(* PLC project Unnamed, Unknown Unnamed 1 *)
(* stored: creationDateTime 2023-09-22T09:24:15, modificationDateTime 2023-09-28T21:40:20 *)

PROGRAM program3
  VAR
    FactoryIOReset0 AT %IX100.0 : BOOL;
    StartButton0 AT %IX100.1 : BOOL;
    EStop0 AT %IX100.2 : BOOL;
    Retro0 AT %IX100.3 : BOOL;
    Retro1 AT %IX100.4 : BOOL;
    VS00 AT %IX100.5 : BOOL;
    VS01 AT %IX100.6 : BOOL;
    VS02 AT %IX100.7 : BOOL;
    VS03 AT %IX101.0 : BOOL;
    TAPP0_Detected AT %IX101.1 : BOOL;
    TAPP0_MovingX AT %IX101.2 : BOOL;
    TAPP0_MovingZ AT %IX101.3 : BOOL;
    TAPP0_Rotating AT %IX101.4 : BOOL;
    Retro2 AT %IX101.5 : BOOL;
    RetroreflectiveSensor3 AT %IX101.6 : BOOL;
    Retro4 AT %IX101.7 : BOOL;
    VS10 AT %IX102.0 : BOOL;
    VS11 AT %IX102.1 : BOOL;
    VS12 AT %IX102.2 : BOOL;
    VisionSensor13 AT %IX102.3 : BOOL;
    TAPP1_Detected AT %IX102.4 : BOOL;
    TwoAxisPickPlace1_MovingX AT %IX102.5 : BOOL;
    TwoAxisPickPlace1_MovingZ AT %IX102.6 : BOOL;
    TwoAxisPickPlace1_Rotating AT %IX102.7 : BOOL;
    RetroreflectiveSensor5 AT %IX103.0 : BOOL;
    RetroreflectiveSensor6 AT %IX103.1 : BOOL;
    Retro7 AT %IX103.2 : BOOL;
    VS20 AT %IX103.3 : BOOL;
    VS21 AT %IX103.4 : BOOL;
    VS22 AT %IX103.5 : BOOL;
    VisionSensor23 AT %IX103.6 : BOOL;
    TAPP2_Detected AT %IX103.7 : BOOL;
    TwoAxisPickPlace2_MovingX AT %IX104.0 : BOOL;
    TwoAxisPickPlace2_MovingZ AT %IX104.1 : BOOL;
    TwoAxisPickPlace2_Rotating AT %IX104.2 : BOOL;
    RetroreflectiveSensor8 AT %IX104.3 : BOOL;
    RetroreflectiveSensor9 AT %IX104.4 : BOOL;
    RetroreflectiveSensor10 AT %IX104.5 : BOOL;
    VisionSensor30 AT %IX104.6 : BOOL;
    VisionSensor31 AT %IX104.7 : BOOL;
    VisionSensor32 AT %IX105.0 : BOOL;
    VisionSensor33 AT %IX105.1 : BOOL;
    Retro11 AT %IX105.2 : BOOL;
    Retro12 AT %IX105.3 : BOOL;
    Retro13 AT %IX105.4 : BOOL;
    Retro14 AT %IX105.5 : BOOL;
    Retro15 AT %IX105.6 : BOOL;
    Retro16 AT %IX105.7 : BOOL;
    TAPP0X AT %QX100.0 : BOOL;
    TAPP0Z AT %QX100.1 : BOOL;
    TAPP0_Grab AT %QX100.2 : BOOL;
    TAPP0_RotateCW AT %QX100.3 : BOOL;
    TAPP0_RotateCCW AT %QX100.4 : BOOL;
    BC_6m_0 AT %QX100.5 : BOOL;
    BC_6m_1 AT %QX100.6 : BOOL;
    BC_6m_2 AT %QX100.7 : BOOL;
    BC_6m_3 AT %QX101.0 : BOOL;
    BC_6m_4 AT %QX101.1 : BOOL;
    TAPP1X AT %QX101.2 : BOOL;
    TAPP1Z AT %QX101.3 : BOOL;
    TAPP1_Grab AT %QX101.4 : BOOL;
    TAPP1_RotateCCW AT %QX101.5 : BOOL;
    TAPP1_RotateCW AT %QX101.6 : BOOL;
    GreenBoxDetected AT %QX101.7 : BOOL;
    TAPP2X AT %QX102.0 : BOOL;
    TAPP2Z AT %QX102.1 : BOOL;
    TAPP2_Grab AT %QX102.2 : BOOL;
    TAPP2_RotateCW AT %QX102.3 : BOOL;
    TAPP2_RotateCCW AT %QX102.4 : BOOL;
    BC_2m_0 AT %QX102.5 : BOOL;
    BlueBoxDetected AT %QX102.6 : BOOL;
    GreyBoxDetected0 AT %QX102.7 : BOOL;
    StackLight0_Green AT %QX103.0 : BOOL;
    StackLight0_Yellow AT %QX103.1 : BOOL;
    StackLight0_Red AT %QX103.2 : BOOL;
    StackLight1_Green AT %QX103.3 : BOOL;
    StackLight1_Yellow AT %QX103.4 : BOOL;
    StackLight1_Red AT %QX103.5 : BOOL;
    StackLight2_Green AT %QX103.6 : BOOL;
    StackLight2_Yellow AT %QX103.7 : BOOL;
    StackLight2_Red AT %QX104.0 : BOOL;
    LightIndicator_Red_2 AT %QX104.1 : BOOL;
    BlueGrabbed AT %QW100 : INT;
    GreenGrabbed AT %QW101 : INT;
    GreyGrabbed AT %QW102 : INT;
    BlueMissed AT %QW103 : INT;
    GreenMissed AT %QW104 : INT;
    GreyMissed AT %QW105 : INT;
  END_VAR
  VAR
    FactoryReset : BOOL;
    StartCondition : BOOL;
    RS1 : RS;
    TAPP0ZPT : TIME := T#2s;
    RCW0PT : TIME := T#2s;
    RCW1PT : TIME := T#2s;
    RCW2PT : TIME := T#2s;
    TAPP1ZPT : TIME := T#2s;
    TAPP2ZPT : TIME := T#2s;
    TAPP0ZET : TIME;
    TAPP1ZET : TIME;
    TAPP2ZET : TIME;
    Grab0PT : TIME := T#0.5s;
    Grab2PT : TIME := T#0.5s;
    Grab1PT : TIME := T#0.5s;
    Grab0ET : TIME;
    RCW0ET : TIME;
    RCW1ET : TIME;
    RCW2ET : TIME;
    Grab1ET : TIME;
    Grab2ET : TIME;
    Grab0TPPT : TIME := T#3s;
    Grab1TPPT : TIME := T#3s;
    Grab2TPPT : TIME := T#3s;
    Grab0TPET : TIME;
    Grab1TPET : TIME;
    Grab2TPET : TIME;
    GreyBox : BOOL;
    RS5 : RS;
    GrabbedMax : INT := 50;
    RS11 : RS;
    RS9 : RS;
    RS10 : RS;
    RS12 : RS;
    TON0 : TON;
    RS14 : RS;
    TON1 : TON;
    RS15 : RS;
    RS16 : RS;
    TON2 : TON;
    TP0 : TP;
    RS13 : RS;
    RS17 : RS;
    RS18 : RS;
    RS2 : RS;
    CTU0 : CTU;
    RS20 : RS;
    CTU1 : CTU;
    RS21 : RS;
    CTU2 : CTU;
    RS30 : RS;
    CTU3 : CTU;
    RS31 : RS;
    RS32 : RS;
    RS7 : RS;
    RS37 : RS;
    RS38 : RS;
    TON8 : TON;
    CTU4 : CTU;
    RS41 : RS;
    CTU5 : CTU;
    RS42 : RS;
    RS19 : RS;
    RS22 : RS;
    RS23 : RS;
    RS24 : RS;
    RS25 : RS;
    TON3 : TON;
    RS6 : RS;
    RS26 : RS;
    RS27 : RS;
    TON4 : TON;
    TP1 : TP;
    TON5 : TON;
    RS28 : RS;
    RS29 : RS;
    RS33 : RS;
    RS34 : RS;
    RS35 : RS;
    RS36 : RS;
    TON6 : TON;
    TP2 : TP;
    TON7 : TON;
    RS43 : RS;
    RS44 : RS;
  END_VAR
  VAR  (* added by the conversion: wires and edge detectors of the diagram *)
    R_TRIG1 : R_TRIG;
    F_TRIG2 : F_TRIG;
    F_TRIG3 : F_TRIG;
    R_TRIG4 : R_TRIG;
    R_TRIG5 : R_TRIG;
    F_TRIG6 : F_TRIG;
    R_TRIG7 : R_TRIG;
    R_TRIG8 : R_TRIG;
    F_TRIG9 : F_TRIG;
    R_TRIG10 : R_TRIG;
    R_TRIG11 : R_TRIG;
  END_VAR

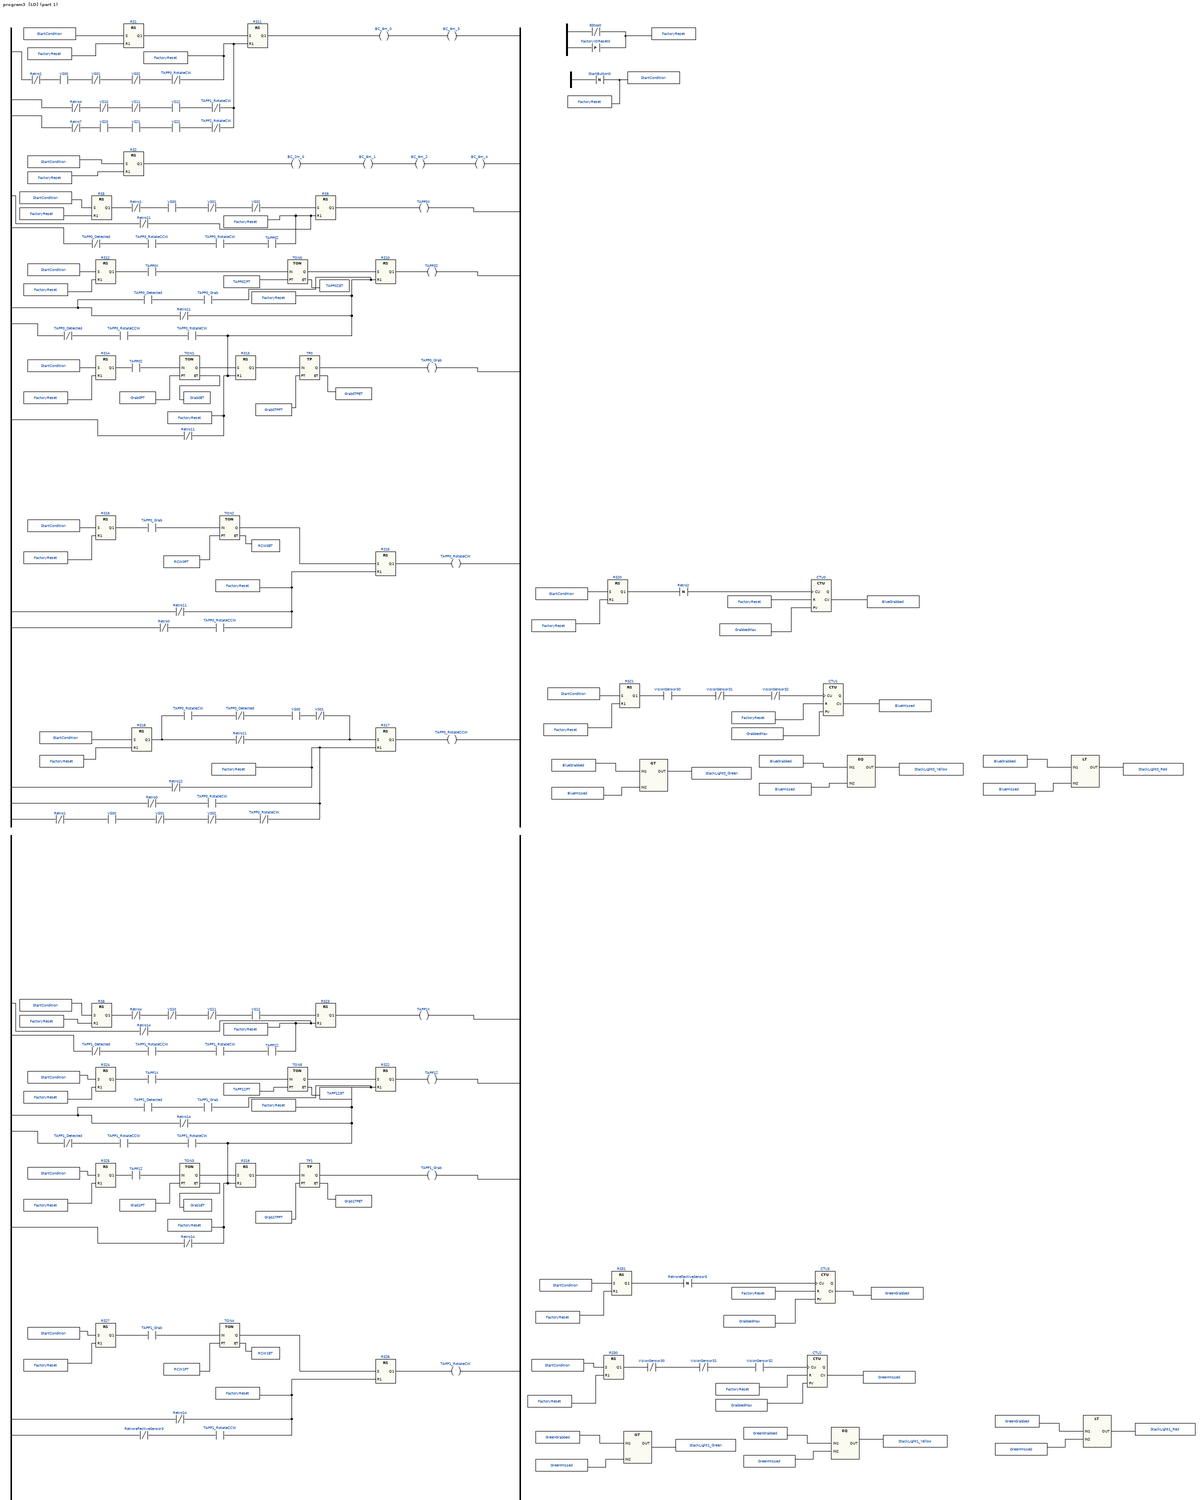
(* LD diagram, written out as Structured Text *)
R_TRIG1(CLK := FactoryIOReset0);
FactoryReset := NOT EStop0 OR R_TRIG1.Q;
RS1(S := StartCondition, R1 := FactoryReset);
RS11(S := RS1.Q1, R1 := FactoryReset OR NOT Retro1 AND VS00 AND NOT VS01 AND NOT VS02 AND NOT TAPP0_RotateCW OR NOT Retro4 AND NOT VS10 AND NOT VS11 AND VS12 AND NOT TAPP1_RotateCW OR NOT Retro7 AND VS20 AND VS21 AND VS22 AND NOT TAPP2_RotateCW);
BC_6m_0 := RS11.Q1;
BC_6m_3 := RS11.Q1;
F_TRIG2(CLK := StartButton0);
StartCondition := F_TRIG2.Q OR FactoryReset;
RS2(S := StartCondition, R1 := FactoryReset);
BC_2m_0 := RS2.Q1;
BC_6m_1 := RS2.Q1;
BC_6m_2 := RS2.Q1;
BC_6m_4 := RS2.Q1;
RS5(S := StartCondition, R1 := FactoryReset);
RS9(S := RS5.Q1 AND NOT Retro1 AND VS00 AND NOT VS01 AND NOT VS02, R1 := FactoryReset OR NOT Retro11 OR NOT TAPP0_Detected AND TAPP0_RotateCCW AND TAPP0_RotateCW AND TAPP0Z);
TAPP0X := RS9.Q1;
RS12(S := StartCondition, R1 := FactoryReset);
TON0(IN := RS12.Q1 AND TAPP0X, PT := TAPP0ZPT);
RS10(S := TON0.Q, R1 := FactoryReset OR TAPP0_Detected AND TAPP0_Grab OR NOT Retro11 OR NOT TAPP0_Detected AND TAPP0_RotateCCW AND TAPP0_RotateCW);
TAPP0Z := RS10.Q1;
TAPP0ZET := TON0.ET;
RS14(S := StartCondition, R1 := FactoryReset);
TON1(IN := RS14.Q1 AND TAPP0Z, PT := Grab0PT);
RS13(S := TON1.Q, R1 := FactoryReset OR NOT Retro11 OR NOT TAPP0_Detected AND TAPP0_RotateCCW AND TAPP0_RotateCW);
TP0(IN := RS13.Q1, PT := Grab0TPPT);
TAPP0_Grab := TP0.Q;
Grab0TPET := TP0.ET;
Grab0ET := TON1.ET;
RS16(S := StartCondition, R1 := FactoryReset);
TON2(IN := RS16.Q1 AND TAPP0_Grab, PT := RCW0PT);
RCW0ET := TON2.ET;
RS15(S := TON2.Q, R1 := FactoryReset OR NOT Retro11 OR NOT Retro0 AND TAPP0_RotateCCW);
TAPP0_RotateCW := RS15.Q1;
RS20(S := StartCondition, R1 := FactoryReset);
F_TRIG3(CLK := Retro2);
R_TRIG4(CLK := RS20.Q1 AND F_TRIG3.Q);
CTU0(CU := R_TRIG4.Q, R := FactoryReset, PV := GrabbedMax);
BlueGrabbed := CTU0.CV;
RS21(S := StartCondition, R1 := FactoryReset);
R_TRIG5(CLK := RS21.Q1 AND VisionSensor30 AND NOT VisionSensor31 AND NOT VisionSensor32);
CTU1(CU := R_TRIG5.Q, R := FactoryReset, PV := GrabbedMax);
BlueMissed := CTU1.CV;
RS18(S := StartCondition, R1 := FactoryReset);
RS17(S := RS18.Q1 AND (NOT Retro11 OR TAPP0_RotateCW AND NOT TAPP0_Detected AND VS00 AND NOT VS01), R1 := FactoryReset OR NOT Retro12 OR NOT Retro1 AND VS00 AND NOT VS01 AND NOT VS02 AND NOT TAPP0_RotateCW OR NOT Retro0 AND TAPP0_RotateCW);
TAPP0_RotateCCW := RS17.Q1;
StackLight0_Yellow := BlueGrabbed = BlueMissed;
StackLight0_Red := BlueGrabbed < BlueMissed;
StackLight0_Green := BlueGrabbed > BlueMissed;
RS6(S := StartCondition, R1 := FactoryReset);
RS23(S := RS6.Q1 AND NOT Retro4 AND NOT VS10 AND NOT VS11 AND VS12, R1 := FactoryReset OR NOT Retro14 OR NOT TAPP1_Detected AND TAPP1_RotateCCW AND TAPP1_RotateCW AND TAPP1Z);
TAPP1X := RS23.Q1;
RS24(S := StartCondition, R1 := FactoryReset);
TON5(IN := RS24.Q1 AND TAPP1X, PT := TAPP1ZPT);
RS22(S := TON5.Q, R1 := FactoryReset OR TAPP1_Detected AND TAPP1_Grab OR NOT Retro14 OR NOT TAPP1_Detected AND TAPP1_RotateCCW AND TAPP1_RotateCW);
TAPP1Z := RS22.Q1;
TAPP1ZET := TON5.ET;
RS25(S := StartCondition, R1 := FactoryReset);
TON3(IN := RS25.Q1 AND TAPP1Z, PT := Grab1PT);
RS19(S := TON3.Q, R1 := FactoryReset OR NOT Retro14 OR NOT TAPP1_Detected AND TAPP1_RotateCCW AND TAPP1_RotateCW);
TP1(IN := RS19.Q1, PT := Grab1TPPT);
TAPP1_Grab := TP1.Q;
Grab1TPET := TP1.ET;
Grab1ET := TON3.ET;
RS31(S := StartCondition, R1 := FactoryReset);
F_TRIG6(CLK := RetroreflectiveSensor5);
R_TRIG7(CLK := RS31.Q1 AND F_TRIG6.Q);
CTU3(CU := R_TRIG7.Q, R := FactoryReset, PV := GrabbedMax);
GreenGrabbed := CTU3.CV;
RS27(S := StartCondition, R1 := FactoryReset);
TON4(IN := RS27.Q1 AND TAPP1_Grab, PT := RCW1PT);
RCW1ET := TON4.ET;
RS26(S := TON4.Q, R1 := FactoryReset OR NOT Retro14 OR NOT RetroreflectiveSensor3 AND TAPP1_RotateCCW);
TAPP1_RotateCW := RS26.Q1;
RS30(S := StartCondition, R1 := FactoryReset);
R_TRIG8(CLK := RS30.Q1 AND NOT VisionSensor30 AND NOT VisionSensor31 AND VisionSensor32);
CTU2(CU := R_TRIG8.Q, R := FactoryReset, PV := GrabbedMax);
GreenMissed := CTU2.CV;
StackLight1_Red := GreenGrabbed < GreenMissed;
StackLight1_Yellow := GreenGrabbed = GreenMissed;
StackLight1_Green := GreenGrabbed > GreenMissed;
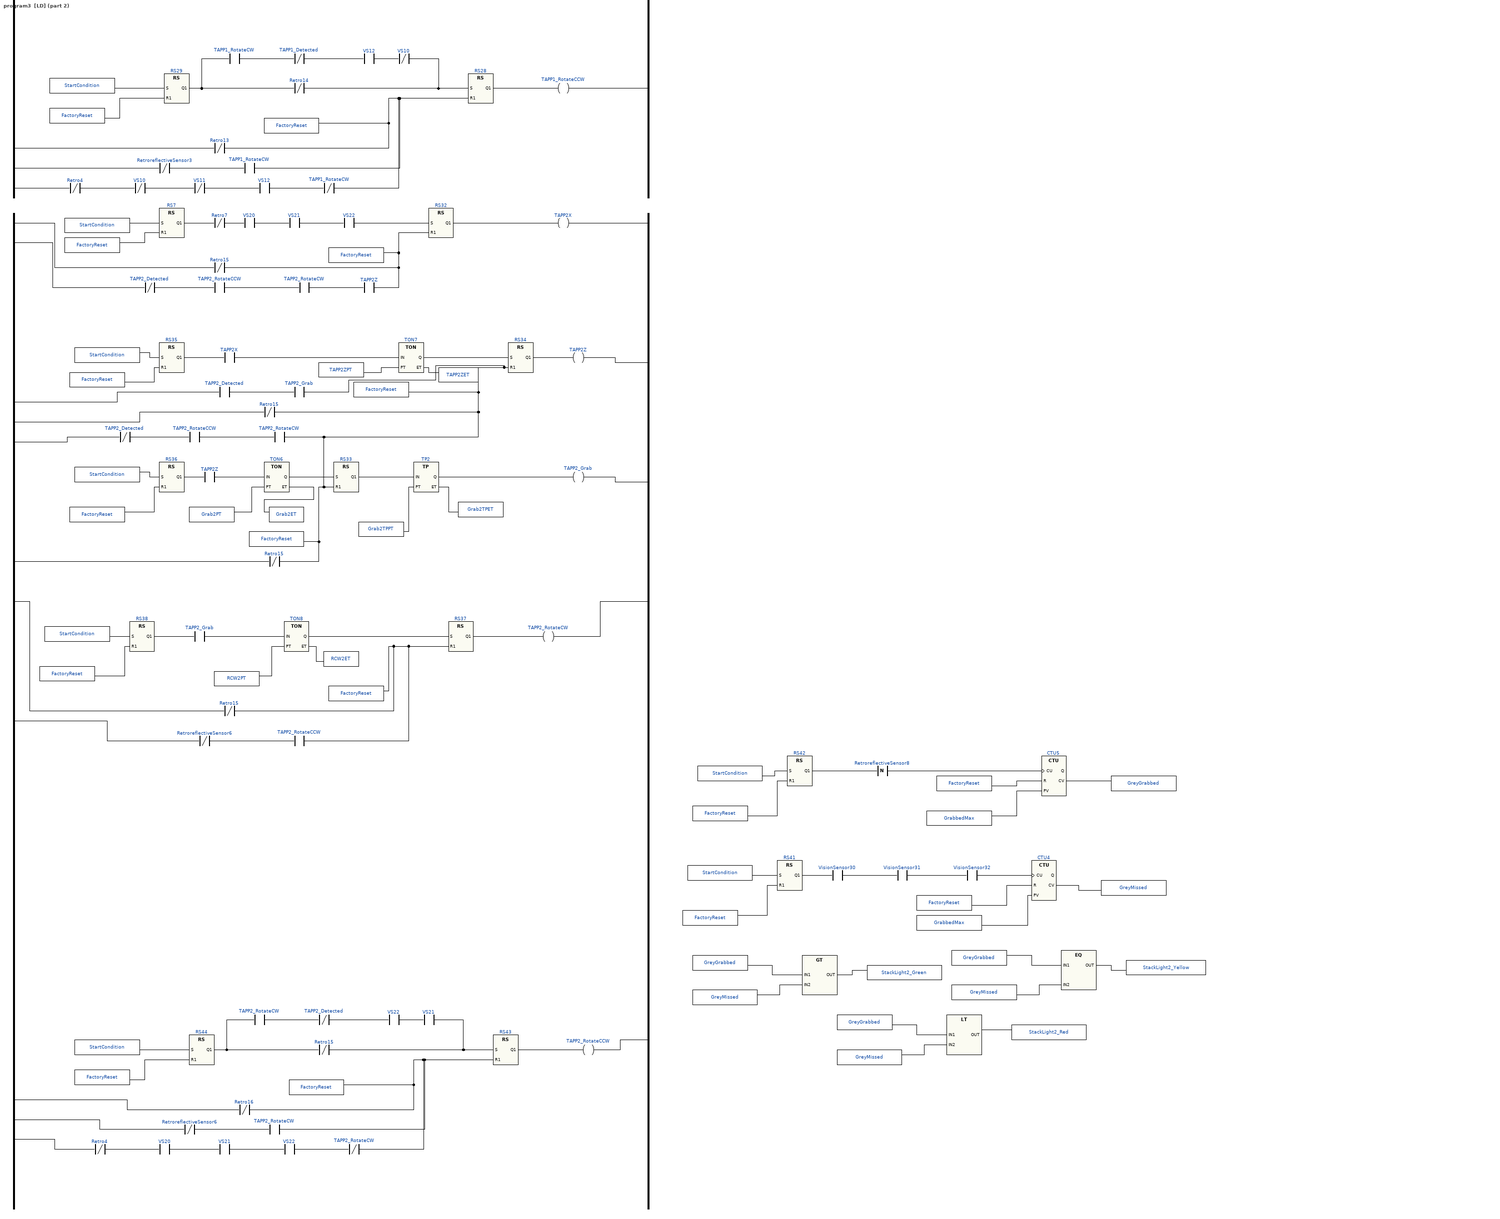
RS29(S := StartCondition, R1 := FactoryReset);
RS28(S := RS29.Q1 AND (NOT Retro14 OR TAPP1_RotateCW AND NOT TAPP1_Detected AND VS12 AND NOT VS10), R1 := FactoryReset OR NOT Retro13 OR NOT Retro4 AND NOT VS10 AND NOT VS11 AND VS12 AND NOT TAPP1_RotateCW OR NOT RetroreflectiveSensor3 AND TAPP1_RotateCW);
TAPP1_RotateCCW := RS28.Q1;
RS7(S := StartCondition, R1 := FactoryReset);
RS32(S := RS7.Q1 AND NOT Retro7 AND VS20 AND VS21 AND VS22, R1 := FactoryReset OR NOT Retro15 OR NOT TAPP2_Detected AND TAPP2_RotateCCW AND TAPP2_RotateCW AND TAPP2Z);
TAPP2X := RS32.Q1;
RS35(S := StartCondition, R1 := FactoryReset);
TON7(IN := RS35.Q1 AND TAPP2X, PT := TAPP2ZPT);
RS34(S := TON7.Q, R1 := FactoryReset OR TAPP2_Detected AND TAPP2_Grab OR NOT Retro15 OR NOT TAPP2_Detected AND TAPP2_RotateCCW AND TAPP2_RotateCW);
TAPP2Z := RS34.Q1;
TAPP2ZET := TON7.ET;
RS36(S := StartCondition, R1 := FactoryReset);
TON6(IN := RS36.Q1 AND TAPP2Z, PT := Grab2PT);
RS33(S := TON6.Q, R1 := FactoryReset OR NOT Retro15 OR NOT TAPP2_Detected AND TAPP2_RotateCCW AND TAPP2_RotateCW);
TP2(IN := RS33.Q1, PT := Grab2TPPT);
TAPP2_Grab := TP2.Q;
Grab2TPET := TP2.ET;
Grab2ET := TON6.ET;
RS38(S := StartCondition, R1 := FactoryReset);
TON8(IN := RS38.Q1 AND TAPP2_Grab, PT := RCW2PT);
RS37(S := TON8.Q, R1 := FactoryReset OR NOT Retro15 OR NOT RetroreflectiveSensor6 AND TAPP2_RotateCCW);
TAPP2_RotateCW := RS37.Q1;
RCW2ET := TON8.ET;
RS42(S := StartCondition, R1 := FactoryReset);
F_TRIG9(CLK := RetroreflectiveSensor8);
R_TRIG10(CLK := RS42.Q1 AND F_TRIG9.Q);
CTU5(CU := R_TRIG10.Q, R := FactoryReset, PV := GrabbedMax);
GreyGrabbed := CTU5.CV;
RS41(S := StartCondition, R1 := FactoryReset);
R_TRIG11(CLK := RS41.Q1 AND VisionSensor30 AND VisionSensor31 AND VisionSensor32);
CTU4(CU := R_TRIG11.Q, R := FactoryReset, PV := GrabbedMax);
GreyMissed := CTU4.CV;
StackLight2_Yellow := GreyGrabbed = GreyMissed;
StackLight2_Green := GreyGrabbed > GreyMissed;
StackLight2_Red := GreyGrabbed < GreyMissed;
RS44(S := StartCondition, R1 := FactoryReset);
RS43(S := RS44.Q1 AND (NOT Retro15 OR TAPP2_RotateCW AND NOT TAPP2_Detected AND VS22 AND VS21), R1 := FactoryReset OR NOT Retro16 OR NOT Retro4 AND VS20 AND VS21 AND VS22 AND NOT TAPP2_RotateCW OR NOT RetroreflectiveSensor6 AND TAPP2_RotateCW);
TAPP2_RotateCCW := RS43.Q1;
END_PROGRAM

CONFIGURATION Config0
  RESOURCE Res0 ON PLC
    TASK task0(INTERVAL := T#20ms, PRIORITY := 0);
    PROGRAM instance0 WITH task0 : program3;
  END_RESOURCE
END_CONFIGURATION
